Universal Robots PolyScope program: URClient.urp

Program URClient (installation=default directory=/home/ur/ursim-current/programs createdIn=3.1.17195 lastSavedIn=5.13.0 robotSerialNumber=20195399999)
Calibrated DH parameters: a=[0, -0.24355, -0.2132, 0, 0, 0]; d=[0.15185, 0, 0, 0.13105, 0.08535, 0.0921]; alpha=[1.570796, 0, 0, 1.570796, -1.570796, 0]; deltaTheta=[0, 0, 0, 0, 0, 0]
InitVariablesNode
BeforeStart
  open := socket_open("192.168.98.23",50000)
  Loop While (checkContinuously=false) expression=open≟ False
    open := socket_open("192.168.98.23",50000)
  Script: socket_send_string("ur_id")
  targetPos := p[0,0,0,0,0,0]
  counter := 0
Robot Program (runOnlyOnce=false)
  Script: socket_send_string("newpose")
  receiveFromServ := socket_read_ascii_float(6)
  Loop While (checkContinuously=false) expression=receiveFromServ[0]≠6
    Wait Sleep waitTime=0.3
    receiveFromServ := socket_read_ascii_float(6)
  Loop While (checkContinuously=false) expression=counter<6
    Script: targetPos[counter]=receiveFromServ[counter+1]
    counter := counter+1
  MoveJ speed 60 deg/s, acceleration 80 deg/s^2 (useActiveTCP=true) feature=Base
    Waypoint Variable (Variable): variable=targetPos
    Wait Sleep waitTime=0.1
  counter := 0
  Script: socket_send_string("urready")
  Wait Sleep waitTime=2
